TYPE ST_PeakShaveBox_Get :
STRUCT
	Powermonitor		: ST_Wago750495_Get;
	Buscoupler			: ST_Wago750354_get;
END_STRUCT
END_TYPE

(* stored: Version 1.1.0.1, ProductVersion 3.1.4024.12
   DUT ST_PeakShaveBox_Get: Id {33c5722f-15da-4d92-854e-828c06ec61ce} *)
